PROGRAM MAIN
VAR
	
i : INT;
couple:bool;
P1: MC_POWER;
Axis1 : AXIS_REF;
P2: MC_POWER;
Axis2 : AXIS_REF;
P3: MC_POWER;
Axis3 : AXIS_REF;
P4: MC_POWER;
Axis4 : AXIS_REF;


M1:DUT_M;
M2:DUT_M;
M3:DUT_M;
M4:DUT_M;

GearIn: MC_GearIn;
GearInOut: ST_McOutputs;
GearOut: MC_GearOut;
GearOutOut: ST_McOutputs;
//X_Axes : FB_Motion();
//Y_Axes : FB_Motion();

x_go: bool;
y_go:bool;
END_VAR

i:=i+1;
//ignore naming lim in and limout
P1(
	Axis:= Axis1 , 
	Enable:= M1.Enable, 
	Enable_Positive:=M1.LimIn AND M1.LimOut , //FFW DI2
	Enable_Negative:= M1.LimOut AND M1.LimIn, 
	Override:= , 
	BufferMode:= , 
	Options:= , 
	Status=> , 
	Busy=> , 
	Active=> , 
	Error=> , 
	ErrorID=> );

P2(
	Axis:= Axis2 , 
	Enable:= M2.Enable, 
	Enable_Positive:=M2.LimIn  , //FFW Di2
	Enable_Negative:= M2.LimOut , 
	Override:= , 
	BufferMode:= , 
	Options:= , 
	Status=> , 
	Busy=> , 
	Active=> , 
	Error=> , 
	ErrorID=> );


P3(
	Axis:= Axis3 , 
	Enable:= M3.Enable, 
	Enable_Positive:= M3.LimOut  ,  //DI1
	Enable_Negative:= M3.LimIn, 
	Override:= , 
	BufferMode:= , 
	Options:= , 
	Status=> , 
	Busy=> , 
	Active=> , 
	Error=> , 
	ErrorID=> );

P4(
	Axis:= Axis4 , 
	Enable:= M4.Enable, 
	Enable_Positive:=M4.LimOut , //DI1
	Enable_Negative:= M4.LimIn, //DI 2 clse to motor fbw cw
	Override:= , 
	BufferMode:= , 
	Options:= , 
	Status=> , 
	Busy=> , 
	Active=> , 
	Error=> , 
	ErrorID=> );
	
Axis1();
Axis2();
Axis3();
Axis4();

(*
if couple then
	GearIn.Execute := TRUE;
	couple:=false;
	IF GearIn.InGear THEN
				GearIn.Execute := FALSE;
			ELSIF GearIn.Error THEN
				//state := MOVESTATE_ERROR;
			END_IF
END_IF
	
//GearOut(
		
ActCouple();
GearIn.RatioNumerator :=1;
GearIn.RatioDenominator :=1;

X_Axes(Master:= Axis3, Slave:=Axis4, PowerMaster:=P3, PowerSlave:=P4, GO:= x_go);
Y_Axes(Master:= Axis1, Slave:=Axis2, PowerMaster:=P1, PowerSlave:=P2, GO:= y_go);*)

ACTION ActCouple:
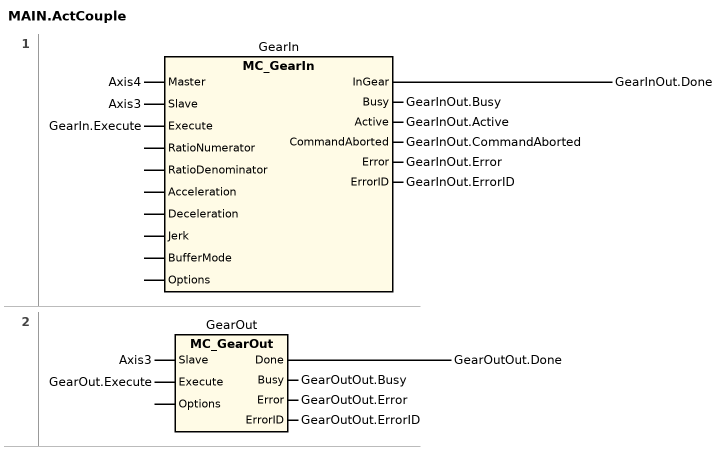
// NETWORK 1
GearIn(
    Master := Axis4,
    Slave := Axis3,
    Execute := GearIn.Execute,
    Busy => GearInOut.Busy,
    Active => GearInOut.Active,
    CommandAborted => GearInOut.CommandAborted,
    Error => GearInOut.Error,
    ErrorID => GearInOut.ErrorID); // MC_GearIn
GearInOut.Done := GearIn.InGear;

// NETWORK 2
GearOut(
    Slave := Axis3,
    Execute := GearOut.Execute,
    Busy => GearOutOut.Busy,
    Error => GearOutOut.Error,
    ErrorID => GearOutOut.ErrorID); // MC_GearOut
GearOutOut.Done := GearOut.Done;
END_ACTION

END_PROGRAM

(* stored: Version 1.1.0.1, ProductVersion 3.1.4024.3
   POU MAIN: Id {8e638a08-55a7-4307-a06b-7186a42625dc}, SpecialFunc None
   Action ActCouple: Id {c7e30986-e2c1-4fb8-b13e-8fca653a147d} *)
